Staubli VAL3: getTool.pgx

public program getTool(tool& x_tTool[], num x_nIndex)
begin
  // get the tool
  x_tTool=saveData:tData[x_nIndex].tcp
end
